PROGRAM RETURN_LASER
VAR_INPUT

END_VAR

VAR
	TMR_DELAY: TON;
	TMR_DELAY1: TON;
	TMR_DELAY2: TON;
END_VAR


IF SORTER_VAR.TRANSPORT_IDX=0 AND SORTER_VAR.STATION_RETURN_IDX=0 AND SORTER_VAR.JIG_RETURN_IDX=0 THEN
	SORTER_VAR.TRANSPORT_IDX:=SORTER_VAR.I_CURRENT_TRANSACTION.TRANSPORT_INDEX;
	SORTER_VAR.STATION_RETURN_IDX:=SORTER_VAR.I_CURRENT_TRANSACTION.STATION_NUMBER_LOAD;
	SORTER_VAR.JIG_RETURN_IDX:=SORTER_VAR.I_CURRENT_TRANSACTION.JIG_INDEX_LOAD;
ELSE
CASE SORTER_VAR.I_CASE OF
0: //standby near lotbox
	IF SORTER_VAR.ACTIVE_ID=6 THEN
		SORTER_VAR.ACTIVE_ID:=1;
	END_IF
	SORTER_VAR.TRANSPORT_IDX:=SORTER_VAR.I_CURRENT_TRANSACTION.TRANSPORT_INDEX;
	SORTER_VAR.STATION_RETURN_IDX:=SORTER_VAR.I_CURRENT_TRANSACTION.STATION_NUMBER_RETURN;
	SORTER_VAR.JIG_RETURN_IDX:=SORTER_VAR.I_CURRENT_TRANSACTION.JIG_INDEX_RETURN;
	CASE SORTER_VAR.I_CURRENT_TRANSACTION.TRANSPORT_INDEX OF
		2 : 
			SORTER_VAR.O_STOPPER_TRANSFER_B:=FALSE;			
			LASER_MOVE(STEP_DATA_1:=0,//3,
				STEP_DATA_2:=0,
				STEP_DATA_3:=12,
				STEP_DATA_4:=0,
				STEP_DATA_5:=1);
				SORTER_VAR.I_RETURN_DONE_B:=FALSE;
		1 : 
			SORTER_VAR.O_STOPPER_TRANSFER_A:=FALSE;
			LASER_MOVE(STEP_DATA_1:=0,//3,
				STEP_DATA_2:=0,
				STEP_DATA_3:=12,
				STEP_DATA_4:=1,
				STEP_DATA_5:=0);
				SORTER_VAR.I_RETURN_DONE_A:=FALSE;
	END_CASE			
	SORTER_VAR.O_VACUUM_On:=FALSE;
	SORTER_VAR.O_VACUUM_OFF:=FALSE;	
	TMR_DELAY(IN:=FALSE);
	SORTER_VAR.O_CARTESSIAN_GRIPPER_ON:=FALSE;
	SORTER_VAR.O_CARTESSIAN_GRIPPER_OFF:=TRUE;

1://ready for picking up
	IF SORTER_VAR.ACTIVE_ID=6 THEN
		SORTER_VAR.ACTIVE_ID:=1;
	END_IF
	SORTER_VAR.O_NG_BUFFER_ON:=TRUE;
	SORTER_VAR.O_NG_BUFFER_OFF:=FALSE;
	CASE SORTER_VAR.TRANSPORT_IDX OF
	1:
		SORTER_VAR.I_RETURN_DONE_A:=FALSE;
		IF NOT SORTER_VAR.I_LASER_TRANSFER_AT_BACK_A THEN
			SORTER_VAR.I_CASE:=0;
		ELSE
			LASER_MOVE(STEP_DATA_1:=0,
				STEP_DATA_2:=1,
				STEP_DATA_3:=11,
				STEP_DATA_4:=1,
				STEP_DATA_5:=0);	
		END_IF
	2:
		SORTER_VAR.I_RETURN_DONE_B:=FALSE;
		IF NOT SORTER_VAR.I_LASER_TRANSFER_AT_BACK_B THEN
			SORTER_VAR.I_CASE:=0;
		ELSE
			LASER_MOVE(STEP_DATA_1:=0,
				STEP_DATA_2:=1,
				STEP_DATA_3:=11,
				STEP_DATA_4:=0,
				STEP_DATA_5:=1);	
		END_IF
	END_CASE
2://ready for picking up
	IF SORTER_VAR.ACTIVE_ID=6 THEN
		SORTER_VAR.ACTIVE_ID:=1;
	END_IF

	CASE SORTER_VAR.TRANSPORT_IDX OF
	1:		
				
//IF SORTER_VAR.I_LASER_TRANSFER_AT_BACK_A THEN
		LASER_MOVE(STEP_DATA_1:=SORTER_VAR.TRANSPORT_IDX+5,
				STEP_DATA_2:=1,
				STEP_DATA_3:=18,
				STEP_DATA_4:=0,
				STEP_DATA_5:=0);
		//END_IF
	2:
		//IF SORTER_VAR.I_LASER_TRANSFER_AT_BACK_B THEN
		//IF  NOT SORTER_VAR.I_LASER_TRANSFER_AT_BACK_B THEN
		LASER_MOVE(STEP_DATA_1:=SORTER_VAR.TRANSPORT_IDX+5,
				STEP_DATA_2:=1,
				STEP_DATA_3:=18,
				STEP_DATA_4:=0,
				STEP_DATA_5:=0);
		//END_IF
	END_CASE

		
3://VACUUM AND TAKEUP
	IF SORTER_VAR.ACTIVE_ID=6 THEN
		SORTER_VAR.ACTIVE_ID:=1;
	END_IF

			LASER_MOVE(STEP_DATA_1:=SORTER_VAR.TRANSPORT_IDX+5,
				STEP_DATA_2:=2,
				STEP_DATA_3:=11,
				STEP_DATA_4:=0,
				STEP_DATA_5:=0);
	
	SORTER_VAR.O_VACUUM_On:=TRUE;
	SORTER_VAR.O_VACUUM_OFF:=FALSE;
	
4://VACUUM AND TAKEUP
	IF SORTER_VAR.ACTIVE_ID=6 THEN
		SORTER_VAR.ACTIVE_ID:=1;
	END_IF

	LASER_MOVE(STEP_DATA_1:=SORTER_VAR.TRANSPORT_IDX+5,
				STEP_DATA_2:=9,
				STEP_DATA_3:=11,
				STEP_DATA_4:=0,
				STEP_DATA_5:=0);
	SORTER_VAR.O_VACUUM_On:=TRUE;
	SORTER_VAR.O_VACUUM_OFF:=FALSE;
	
5://MOVE BACK 10MM
	IF SORTER_VAR.ACTIVE_ID=6 THEN
		SORTER_VAR.ACTIVE_ID:=1;
	END_IF
	SORTER_VAR.O_CARTESSIAN_GRIPPER_ON:=TRUE;
	SORTER_VAR.O_CARTESSIAN_GRIPPER_OFF:=FALSE;
	IF SORTER_VAR.I_CARTESSIAN_GRIPPER_ON THEN
	LASER_MOVE(STEP_DATA_1:=SORTER_VAR.TRANSPORT_IDX+5,
				STEP_DATA_2:=10,
				STEP_DATA_3:=SORTER_VAR.JIG_RETURN_IDX,//12,
				STEP_DATA_4:=0,
				STEP_DATA_5:=0);
END_IF
		
6://vacuum position 
	IF SORTER_VAR.ACTIVE_ID=6 THEN
		SORTER_VAR.ACTIVE_ID:=1;
	END_IF
	//SORTER_VAR.I_CASE:=SORTER_VAR.I_CASE+1;
	
	TMR_DELAY(IN:=TRUE,PT:=T#1S);
	IF TMR_DELAY.Q THEN
			LASER_MOVE(STEP_DATA_1:=SORTER_VAR.STATION_RETURN_IDX,
				STEP_DATA_2:=3,
				STEP_DATA_3:=14,
				STEP_DATA_4:=0,
				STEP_DATA_5:=0);
	END_IF
				
7://INSERT INTO LOTBOX
	IF SORTER_VAR.ACTIVE_ID=6 THEN
		SORTER_VAR.ACTIVE_ID:=1;
	END_IF
	TMR_DELAY(IN:=FALSE);
	LASER_MOVE(STEP_DATA_1:=SORTER_VAR.STATION_RETURN_IDX,
				STEP_DATA_2:=4,
				STEP_DATA_3:=SORTER_VAR.JIG_RETURN_IDX,//16,
				STEP_DATA_4:=0,
				STEP_DATA_5:=0);
				
8://MOVE BACK
	IF SORTER_VAR.ACTIVE_ID=6 THEN
		SORTER_VAR.ACTIVE_ID:=1;
	END_IF
	TMR_DELAY2 (IN:=TRUE,PT:=T#2S);
	//IF TMR_DELAY2.Q THEN
	SORTER_VAR.O_CARTESSIAN_GRIPPER_ON:=FALSE;
	SORTER_VAR.O_CARTESSIAN_GRIPPER_OFF:=TRUE;
	IF SORTER_VAR.I_CARTESSIAN_GRIPPER_OFF THEN
		LASER_MOVE(STEP_DATA_1:=SORTER_VAR.STATION_RETURN_IDX,
				STEP_DATA_2:=10,
				STEP_DATA_3:=18,//SORTER_VAR.I_CURRENT_TRANSACTION.JIG_INDEX_RETURN,
				STEP_DATA_4:=0,
				STEP_DATA_5:=0);
	END_IF
	SORTER_VAR.O_VACUUM_On:=FALSE;
	SORTER_VAR.O_VACUUM_OFF:=TRUE;
9: //standby near lotbox
	
	IF SORTER_VAR.ACTIVE_ID=6 THEN
		SORTER_VAR.ACTIVE_ID:=1;
	END_IF
	//SORTER_VAR.I_CASE:=SORTER_VAR.I_CASE+1;
	LASER_MOVE(STEP_DATA_1:=SORTER_VAR.STATION_RETURN_IDX,
				STEP_DATA_2:=1,
				STEP_DATA_3:=10,//SORTER_VAR.I_CURRENT_TRANSACTION.JIG_INDEX_RETURN,
				STEP_DATA_4:=0,
				STEP_DATA_5:=0);

				
10://vacuum position 
	IF SORTER_VAR.ACTIVE_ID=6 THEN
		SORTER_VAR.ACTIVE_ID:=1;
	END_IF
	LASER_MOVE(STEP_DATA_1:=0,
				STEP_DATA_2:=1,
				STEP_DATA_3:=4,
				STEP_DATA_4:=0,
				STEP_DATA_5:=0);
	IF SORTER_VAR.ACTIVE_ID=3 THEN
		SORTER_VAR.O_VACUUM_ON:=FALSE;
		SORTER_VAR.O_VACUUM_OFF:=FALSE;	
	END_IF
		
100:
	SORTER_VAR.O_NG_BUFFER_ON:=FALSE;
	SORTER_VAR.O_NG_BUFFER_OFF:=FALSE;
	SORTER_VAR.O_VACUUM_On:=FALSE;
	SORTER_VAR.O_VACUUM_OFF:=FALSE;
END_CASE 
END_IF
IF SORTER_VAR.I_CASE=11 THEN
			CASE SORTER_VAR.TRANSPORT_IDX OF
		1:
			SORTER_VAR.I_RETURN_DONE_A:=TRUE;
		
		2:
			SORTER_VAR.I_RETURN_DONE_B:=TRUE;
	END_CASE
	IF SORTER_VAR.I_RETURN_DONE_A OR SORTER_VAR.I_RETURN_DONE_B THEN
		FLAG_VAR.ALLOW_EXECUTE_RETURN_LASER:=FALSE;
		TMR_DELAY(IN:=FALSE);
		TMR_DELAY1(IN:=FALSE);
		TMR_DELAY2(IN:=FALSE);
		
		SORTER_VAR.I_CASE:=100;
	END_IF
END_IF

END_PROGRAM

(* stored: Version 1.1.0.1, ProductVersion 3.1.4020.12
   POU RETURN_LASER: Id {1114e93a-06c3-45fb-a632-c3bb59274df1}, SpecialFunc None *)
